	//iFinalVeloContactCaseAdv
		aTransferPackages[25].iChannel := iParameterSet;
		aTransferPackages[25].iAddressedTarget := 33;
		aTransferPackages[25].iIndex := 156;
		
	//iMeanPressureLevel
		aTransferPackages[26].iChannel := iParameterSet;
		aTransferPackages[26].iAddressedTarget := 33;
		aTransferPackages[26].iIndex := 184;
		
	// iThreshPosFollowError
		aTransferPackages[27].iChannel := iParameterSet;
		aTransferPackages[27].iAddressedTarget := 33;
		aTransferPackages[27].iIndex := 204;
		
	// iTreshVeloFollowError
		aTransferPackages[28].iChannel := iParameterSet;
		aTransferPackages[28].iAddressedTarget := 33;
		aTransferPackages[28].iIndex := 205;
		
	// iSoftStartFunction
		aTransferPackages[29].iChannel := iParameterSet;
		aTransferPackages[29].iAddressedTarget := 33;
		aTransferPackages[29].iIndex := 222;
		
	// iEndPositionMonitoring
		aTransferPackages[30].iChannel := iParameterSet;
		aTransferPackages[30].iAddressedTarget := 33;
		aTransferPackages[30].iIndex := 224;
		
	// xOptionPressureBuildUpIntoMechEndPos
		aTransferPackages[31].iChannel := iParameterSet;
		aTransferPackages[31].iAddressedTarget := 33;
		aTransferPackages[31].iIndex := 225;
		
	// iOptControllerGainRelative
		aTransferPackages[32].iChannel := iParameterSet;
		aTransferPackages[32].iAddressedTarget := 33;
		aTransferPackages[32].iIndex := 230;
		
	// iOptDampingOfSystemAbsolute
		aTransferPackages[33].iChannel := iParameterSet;
		aTransferPackages[33].iAddressedTarget := 33;
		aTransferPackages[33].iIndex := 231;
		
	// iOptPliabilityRelative
		aTransferPackages[34].iChannel := iParameterSet;
		aTransferPackages[34].iAddressedTarget := 33;
		aTransferPackages[34].iIndex := 232;
		
	// iOptReductionOfPilotControlRelative
		aTransferPackages[35].iChannel := iParameterSet;
		aTransferPackages[35].iAddressedTarget := 33;
		aTransferPackages[35].iIndex := 233;
		
	// iOptCoulombFritionInAccountRelative
		aTransferPackages[36].iChannel := iParameterSet;
		aTransferPackages[36].iAddressedTarget := 33;
		aTransferPackages[36].iIndex := 234;
		
	// define end of parameter list to be uploaded by setting all variables to 0 (end criterion for FB_Upload_Multiple_Parameters)
		aTransferPackages[37].iChannel := 0;
		aTransferPackages[37].iAddressedTarget := 0;
		aTransferPackages[37].iIndex := 0;
//-----------------------------------------------------------------------------------------------------------

// Read the current status of the the motion terminal
	fbreadbitsfromword(wData:= awBusDataFromVTEM[0], iStartBit:=0, iEndBit:= 5, iValue=> iCurrentValveMode, xError=> );				// read current valve mode
//-----------------------------------------------------------------------------------------------------------

// Transition: Aborting condition when xAbort is TRUE in all States except "IDLE" , "ABORTING" and "RESETTING"
	IF xAbort = TRUE AND NOT(iState = 10 AND xExecute = FALSE) AND iState <> 80 AND iState <> 100 THEN
		xStateChange := TRUE;	// Leaving current state
		iState := 80;	// Choosing next state, here: ABORTING
	END_IF
//-----------------------------------------------------------------------------------------------------------

// local state machine
	CASE iState OF
		10:	// IDLE
			// code that is executed only in the first cycle of this state
				IF xStateChange = TRUE THEN
					xStateChange := FALSE;
					iResponse := eTransferResponse.ready_for_new_transfer;
					xDone := FALSE;
					xError := FALSE;
					xBusy := FALSE;
					xAborted := FALSE;
				END_IF
			//-----------------------------------------------------------------------------------------------------------
			
			// code that is repeated every cycle in this state
				iCommandNumber := 0;
			//-----------------------------------------------------------------------------------------------------------
			
			// Transition
			IF xExecute = TRUE THEN
				xStateChange := TRUE;
				iState := 20;
			END_IF
			//-----------------------------------------------------------------------------------------------------------
		
		20:	// RESETTING VALVE MODE TO 61
			// code that is executed only in the first cycle of this state
				IF xStateChange = TRUE THEN
					xStateChange := FALSE;
					iResponse := eTransferResponse.preparing_transfer;
					xDone := FALSE;
					xError := FALSE;
					xBusy := TRUE;
					xAborted := FALSE;
				END_IF
			//-----------------------------------------------------------------------------------------------------------
			
			// code that is repeated every cycle in this state	
				IF iCurrentValveMode = 63 THEN
					iCommandNumber := 5;	// exit transfer mode
				ELSIF iCurrentValveMode <> 61 AND iCurrentValveMode <> 63 THEN
					iCommandNumber := 6;	// stop running motion apps
				END_IF 
			//-----------------------------------------------------------------------------------------------------------
			
			// Transition
				IF iCurrentValveMode = 61 THEN
					xStateChange := TRUE;	// Leave this state
					iState := 30;
					iCommandNumber := 30;			
				END_IF
			//-----------------------------------------------------------------------------------------------------------
		
		30:	// READING PARAMETER VALUES
			// code that is executed only in the first cycle of this state
				IF xStateChange = TRUE THEN
					xStateChange := FALSE;
					iResponse := eTransferResponse.transferring;
					xDone := FALSE;
					xError := FALSE;
					xBusy := TRUE;
					xAborted := FALSE;
				END_IF
			//-----------------------------------------------------------------------------------------------------------
			
			// code that is repeated every cycle in this state
				iCommandNumber := 30;		// read parameter values
			//-----------------------------------------------------------------------------------------------------------
			
			// Transition
				IF fbuploadMultipleParameters.xExecute = TRUE AND fbuploadMultipleParameters.xUploadDone = TRUE AND fbuploadMultipleParameters.xUploadError = FALSE THEN	// Upload Done
					xStateChange := TRUE;
					iState := 40;	// Write parameter values to outputs
				ELSIF fbuploadMultipleParameters.xExecute = TRUE AND fbuploadMultipleParameters.xUploadDone = FALSE AND fbuploadMultipleParameters.xUploadError = TRUE THEN	// Error during update
					xStateChange := TRUE;
					iState := 70;	// ERROR
					iResponse := fbuploadMultipleParameters.iResponse;
				END_IF
			//-----------------------------------------------------------------------------------------------------------
		
		40:	// WRITE PARAMETER VALUES TO OUTPUTS
			// code that is executed only in the first cycle of this state
				IF xStateChange = TRUE THEN
					xStateChange := FALSE;
					iResponse := eTransferResponse.transferring;
					xDone := FALSE;
					xError := FALSE;
					xBusy := TRUE;
					xAborted := FALSE;
				END_IF
			//-----------------------------------------------------------------------------------------------------------
			
			// code that is repeated every cycle in this state
				iTubingLengthAt2						:= aTransferPackages[0].iTransferValue;
				iTubingLengthAt4						:= aTransferPackages[1].iTransferValue;
				iTubingInnerDiameterAt2					:= aTransferPackages[2].iTransferValue;
				iTubingInnerDiameterAt4					:= aTransferPackages[3].iTransferValue;
				iDriveType								:= aTransferPackages[4].iTransferValue;
				iDriveStroke							:= aTransferPackages[5].iTransferValue;
				iInstallationPositionDrive				:= aTransferPackages[6].iTransferValue;
				iOffsetAxisZeroPoint					:= aTransferPackages[7].iTransferValue;
				iInPortFullStrokeMeas					:= aTransferPackages[8].iTransferValue;
				iInPortPartStrokeMeasRet				:= aTransferPackages[9].iTransferValue;
				iInPortPartStrokeMeasAdv				:= aTransferPackages[10].iTransferValue;
				iLoad									:= aTransferPackages[11].iTransferValue;
				iDampingTimeForTargetPositionReached	:= aTransferPackages[12].iTransferValue;
				iDurationOfThresholdExceedanceForError	:= aTransferPackages[13].iTransferValue;
				iToleranceForTargetPositionReached		:= aTransferPackages[14].iTransferValue;
				iMaxVelocityGeneral						:= aTransferPackages[15].iTransferValue;
				iMaxAcceleration						:= aTransferPackages[16].iTransferValue;
				iMaxDeceleration						:= aTransferPackages[17].iTransferValue;
				iMaxJerk								:= aTransferPackages[18].iTransferValue;
				iOffsetProjectZeroPoint					:= aTransferPackages[19].iTransferValue;
				iOffsetSoftLimitNegEndRet				:= aTransferPackages[20].iTransferValue;
				iOffsetSoftLimitPosEndAdv				:= aTransferPackages[21].iTransferValue;
				iDistTargPosWithConstVeloRet			:= aTransferPackages[22].iTransferValue;
				iFinalVeloContactCaseRet				:= aTransferPackages[23].iTransferValue;
				iDistTargPosWithConstVeloAdv			:= aTransferPackages[24].iTransferValue;
				iFinalVeloContactCaseAdv				:= aTransferPackages[25].iTransferValue;
				iMeanPressureLevel						:= aTransferPackages[26].iTransferValue;
				iThreshPosFollowError					:= aTransferPackages[27].iTransferValue;
				iTreshVeloFollowError					:= aTransferPackages[28].iTransferValue;
				iSoftStartFunction						:= aTransferPackages[29].iTransferValue;
				iEndPositionMonitoring					:= aTransferPackages[30].iTransferValue;
				xOptionPressureBuildUpIntoMechEndPos	:= INT_TO_BOOL(aTransferPackages[31].iTransferValue);
				iOptControllerGainRelative				:= aTransferPackages[32].iTransferValue;
				iOptDampingOfSystemAbsolute				:= aTransferPackages[33].iTransferValue;
				iOptPliabilityRelative					:= aTransferPackages[34].iTransferValue;
				iOptReductionOfPilotControlRelative		:= aTransferPackages[35].iTransferValue;
				iOptCoulombFritionInAccountRelative		:= aTransferPackages[36].iTransferValue;
			//-----------------------------------------------------------------------------------------------------------
			
			// Transition
				xStateChange := TRUE;
				iState := 50;
				iCommandNumber := 40;
			//-----------------------------------------------------------------------------------------------------------
		
		50:	// DONE
			// code that is executed only in the first cycle of this state
				IF xStateChange = TRUE THEN
					xStateChange := FALSE;
					iResponse := eTransferResponse.transfer_successful;
					xDone := TRUE;
					xError := FALSE;
					xBusy := FALSE;
					xAborted := FALSE;
				END_IF
			//-----------------------------------------------------------------------------------------------------------
			
			// code that is repeated every cycle in this state	
				IF fbuploadMultipleParameters.xExecute = FALSE  AND fbuploadMultipleParameters.xUploadDone = FALSE AND fbuploadMultipleParameters.xUploadError = FALSE AND iCurrentValveMode = 63 THEN		//FB_UploadMultipleParameters was reset
					iCommandNumber := 5;	// exit transfer mode
				END_IF
			//-----------------------------------------------------------------------------------------------------------
			
			// Transition
				IF fbuploadMultipleParameters.xExecute = FALSE  AND fbuploadMultipleParameters.xUploadDone = FALSE AND fbuploadMultipleParameters.xUploadError = FALSE AND xExecute = FALSE THEN
					xStateChange := TRUE;
					iState := 100;
				END_IF
			//-----------------------------------------------------------------------------------------------------------
			
		70:	// ERROR
			// code that is executed only in the first cycle of this state
				IF xStateChange = TRUE THEN
					xStateChange := FALSE;
					//iResponse := eTransferResponse.communication_failed;	// set within the transition of the last state
					xDone := FALSE;
					xError := TRUE;
					xBusy := FALSE;
					xAborted := FALSE;
				END_IF
			//-----------------------------------------------------------------------------------------------------------
			
			// code that is repeated every cycle in this state	
			//-----------------------------------------------------------------------------------------------------------
			
			// Transition
				IF xExecute = FALSE AND xAbort = FALSE THEN
					xStateChange := TRUE;
					iState := 100;
				END_IF
			//-----------------------------------------------------------------------------------------------------------
			
		80:	// ABORTING
			// code that is executed only in the first cycle of this state
				IF xStateChange = TRUE THEN
					xStateChange := FALSE;
					iResponse := eTransferResponse.aborting;
					xBusy := FALSE;
					xDone := FALSE;
					xError := FALSE;
					xAborted := TRUE;
				END_IF
			//-----------------------------------------------------------------------------------------------------------
			
			// code that is repeated every cycle in this state
				IF iCurrentValveMode = 63 THEN
					iCommandNumber := 5;	// exit transfer mode
				ELSIF iCurrentValveMode <> 61 AND iCurrentValveMode <> 63 THEN
					iCommandNumber := 6;	// stop running motion apps
				ELSE
					iCommandNumber := 0; 
				END_IF
			//-----------------------------------------------------------------------------------------------------------
			
			// Transition
				IF xAbort = FALSE AND xExecute = FALSE AND iCurrentValveMode = 61 THEN
					xStateChange := TRUE;
					iState := 100;
				END_IF
			//-----------------------------------------------------------------------------------------------------------

		100:	// RESETTING FUNCTION BLOCK AND VALVE
			// code that is executed only in the first cycle of this state
				IF xStateChange = TRUE THEN
					xStateChange := FALSE;
					iResponse := eTransferResponse.resetting;
					xDone := FALSE;
					xError := FALSE;
					xBusy := FALSE;
					xAborted := FALSE;
				END_IF
			//-----------------------------------------------------------------------------------------------------------
			
			// code that is repeated every cycle in this state	
				IF iCurrentValveMode = 63 THEN
					iCommandNumber := 5;	// exit transfer mode
				ELSIF iCurrentValveMode <> 61 AND iCurrentValveMode <> 63 THEN
					iCommandNumber := 6;	// stop running motion apps
				END_IF
				
				// reset funktion block fbreadmultipleparameters
				// not done via command number because this is used to reset valve
					fbuploadMultipleParameters(
						awBusDataFromVTEM:= awBusDataFromVTEM, 
						awBusDataToVTEM:= awBusDataToVTEM, 
						xExecute:= FALSE, 
						iResponse=> , 
						iCurrentValue=> , 
						xUploadDone=> , 
						xUploadError=> , 
						aTransferPackages:= aTransferPackages);
				
				// reset parameter outputs
					iParameterSet							:= 1;

					iTubingLengthAt2						:= 0;
					iTubingLengthAt4						:= 0;
					iTubingInnerDiameterAt2					:= 0;
					iTubingInnerDiameterAt4					:= 0;
					iDriveType								:= 0;
					iDriveStroke							:= 0;
					iInstallationPositionDrive				:= 0;
					iOffsetAxisZeroPoint					:= 0;
					iInPortFullStrokeMeas					:= 0;
					iInPortPartStrokeMeasRet				:= 0;
					iInPortPartStrokeMeasAdv				:= 0;
					iLoad									:= 0;
					iDampingTimeForTargetPositionReached	:= 0;
					iDurationOfThresholdExceedanceForError	:= 0;
					iToleranceForTargetPositionReached		:= 0;
					iMaxVelocityGeneral						:= 0;
					iMaxAcceleration						:= 0;
					iMaxDeceleration						:= 0;
					iMaxJerk								:= 0;
					iOffsetProjectZeroPoint					:= 0;
					iOffsetSoftLimitNegEndRet				:= 0;
					iOffsetSoftLimitPosEndAdv				:= 0;
					iDistTargPosWithConstVeloRet			:= 0;
					iFinalVeloContactCaseRet				:= 0;
					iDistTargPosWithConstVeloAdv			:= 0;
					iFinalVeloContactCaseAdv				:= 0;
					iMeanPressureLevel						:= 0;
					iThreshPosFollowError					:= 0;
					iTreshVeloFollowError					:= 0;
					iSoftStartFunction						:= 0;
					iEndPositionMonitoring					:= 0;
					xOptionPressureBuildUpIntoMechEndPos	:= 0;
					iOptControllerGainRelative				:= 0;
					iOptDampingOfSystemAbsolute				:= 0;
					iOptPliabilityRelative					:= 0;
					iOptReductionOfPilotControlRelative		:= 0;
					iOptCoulombFritionInAccountRelative		:= 0;
				
				// reset parameter array
					FOR iCounterResetArray := 0 TO 100 BY 1 DO
						aTransferPackages[iCounterResetArray].iChannel := 0;
						aTransferPackages[iCounterResetArray].iAddressedTarget := 0;
						aTransferPackages[iCounterResetArray].iIndex := 0;
						aTransferPackages[iCounterResetArray].iTransferValue := 0;
					END_FOR
					
					iCounterResetArray := 0;
					xFirstCycle := TRUE;
			//-----------------------------------------------------------------------------------------------------------
			
			// Transition
				IF iCurrentValveMode = 61 THEN
					iCommandNumber := 6; // Last command to send before the FB is in IDLE
					xStateChange := TRUE;
					iState := 10;
				END_IF
			//-----------------------------------------------------------------------------------------------------------
			
	END_CASE
//-----------------------------------------------------------------------------------------------------------

// Command section
	CASE iCommandNumber OF
		0:	// IDLE
			;
		
		5:	// EXIT TRANSFER MODE
			fbwritevaluetoword(iValue:=63, iStartBit:=0, iEndBit:=5, wDataWord:=awBusDataToVTEM[0], xError=> );							// Valve Mode = 63
			fbwritevaluetoword(iValue:=0, iStartBit:=6, iEndBit:=7, wDataWord:=awBusDataToVTEM[0], xError=> );							// 0 (unused)
			fbwritevaluetoword(iValue:=0, iStartBit:=8, iEndBit:=12, wDataWord:=awBusDataToVTEM[0], xError=> );							// Channel = 0 (ignored)
			fbwritevaluetoword(iValue:=3, iStartBit:=13, iEndBit:=15, wDataWord:=awBusDataToVTEM[0], xError=> );						// Transfer Control = 3 (Exit transfer mode)
			fbwritevaluetoword(iValue:=0, iStartBit:=0, iEndBit:=7, wDataWord:=awBusDataToVTEM[1], xError=> );							// Addressed Target = 0 (ignored)
			fbwritevaluetoword(iValue:=0, iStartBit:=8, iEndBit:=15, wDataWord:=awBusDataToVTEM[1], xError=> );							// Index = 0 (ignored)
			fbwritevaluetoword(iValue:=0, iStartBit:=0, iEndBit:=15, wDataWord:=awBusDataToVTEM[2], xError=> );							// Value = 0 (ignored)
			
		6:	// STOP RUNNING MOTION APP
			fbwritevaluetoword(iValue:=61, iStartBit:=0, iEndBit:=5, wDataWord:=awBusDataToVTEM[0], xError=> );							// Valve Mode = 61 (stop)
			fbwritevaluetoword(iValue:=0, iStartBit:=6, iEndBit:=7, wDataWord:=awBusDataToVTEM[0], xError=> );							// App Control = 0 (unused)
			fbwritevaluetoword(iValue:=0, iStartBit:=8, iEndBit:=15, wDataWord:=awBusDataToVTEM[0], xError=> );							// App Option = 0 (unused)
			fbwritevaluetoword(iValue:=0, iStartBit:=0, iEndBit:=15, wDataWord:=awBusDataToVTEM[1], xError=> );							// Setpoint Value 1 = 0 (unused)
			fbwritevaluetoword(iValue:=0, iStartBit:=0, iEndBit:=15, wDataWord:=awBusDataToVTEM[2], xError=> );							// Setpoint Value 2 = 0 (unused)
		
		30:	// RUN FB_UPLOADMULTIPLEPARAMETERS
			fbuploadMultipleParameters(
				awBusDataFromVTEM:= awBusDataFromVTEM, 
				awBusDataToVTEM:= awBusDataToVTEM, 
				xExecute:= TRUE, 
				iResponse=> , 
				iCurrentValue=> , 
				xUploadDone=> , 
				xUploadError=> , 
				aTransferPackages:= aTransferPackages);

		40:	// RESET FB_UPLOADMULTIPLEPARAMETERS
			fbuploadMultipleParameters(
				awBusDataFromVTEM:= awBusDataFromVTEM, 
				awBusDataToVTEM:= awBusDataToVTEM, 
				xExecute:= FALSE, 
				iResponse=> , 
				iCurrentValue=> , 
				xUploadDone=> , 
				xUploadError=> , 
				aTransferPackages:= aTransferPackages);
	END_CASE
//-----------------------------------------------------------------------------------------------------------

END_FUNCTION_BLOCK

// Transfermode/FB_Read_config_AI_Module
/// This function block can be used to upload the configuration of the analog input module on the Motion Terminal.
/// The specific parameters of this module are the outputs of this FB
/// The function block uses the transfer mode to read this configuration from the Motion Terminal
/// and indicates the state of the upload process at the output iResponse.

FUNCTION_BLOCK FB_Read_config_AI_Module
VAR_INPUT
	awBusDataFromVTEM 				: ARRAY [0..2] OF WORD;		// array of 3 words of process data received from the Motion Terminal
END_VAR
	
VAR_IN_OUT
	awBusDataToVTEM 				: ARRAY [0..2] OF WORD; 	// array of 3 words of process data sent to the Motion Terminal
END_VAR

VAR_INPUT
	xExecute 						: BOOL; 					// rising edge starts the reading process, falling edge resets the function block after reading is done
	xAbort							: BOOL;						// rising edge aborts the reading process
	iInputModuleNr					: INT;						// Number of the input module, counted from left to right beginning with 1
END_VAR                     		

VAR_OUTPUT                  		
	// sensor parameters
		iSensorTypePort0			: INT;						// ID of the sensor type, that is connected to the port 0 (0 = no sensor, 2001 = SDAP-MHS-M50, 2002 = SDAP-MHS-M100, 2003 = SDAP-MHS-M160, 2901 = custom position sensor 1, 2902 = custom position sensor 2, 2903 = custom position sensor 3, 3001 = SFAB-50U-…-2SA-…, 3002 = SFAB-200U-…-2SA-…, 3003 = SFAB-600U-…-2SA-…, 3004 = SFAB-1000U-…-2SA-…, 3101 = SFAH-50U-…-PNVBA-…, 3102 = SFAH-100U-…-PNVBA-…, 3103 = SFAH-200U-…-PNVBA-…, 3901 = custom flow sensor 1, 3902 = custom flow sensor 2, 3903 = custom flow sensor 3)
		iSensorOrientPort0			: INT;						// Orientation of the sensor that is connected to the port 0 (position sensor: 0 = risigng current level when advancing, 1 = falling current level when advancing; flow sensor: 0 = positive flow rate values "blowing", 1 = negative flow rate values "drawning")
		iSensorTypePort1			: INT;						// ID of the sensor type, that is connected to the port 1 (0 = no sensor, 2001 = SDAP-MHS-M50, 2002 = SDAP-MHS-M100, 2003 = SDAP-MHS-M160, 2901 = custom position sensor 1, 2902 = custom position sensor 2, 2903 = custom position sensor 3, 3001 = SFAB-50U-…-2SA-…, 3002 = SFAB-200U-…-2SA-…, 3003 = SFAB-600U-…-2SA-…, 3004 = SFAB-1000U-…-2SA-…, 3101 = SFAH-50U-…-PNVBA-…, 3102 = SFAH-100U-…-PNVBA-…, 3103 = SFAH-200U-…-PNVBA-…, 3901 = custom flow sensor 1, 3902 = custom flow sensor 2, 3903 = custom flow sensor 3)
		iSensorOrientPort1			: INT;						// Orientation of the sensor that is connected to the port 0 (position sensor: 0 = risigng current level when advancing, 1 = falling current level when advancing; flow sensor: 0 = positive flow rate values "blowing", 1 = negative flow rate values "drawning")
		iSensorTypePort2			: INT;						// ID of the sensor type, that is connected to the port 2 (0 = no sensor, 2001 = SDAP-MHS-M50, 2002 = SDAP-MHS-M100, 2003 = SDAP-MHS-M160, 2901 = custom position sensor 1, 2902 = custom position sensor 2, 2903 = custom position sensor 3, 3001 = SFAB-50U-…-2SA-…, 3002 = SFAB-200U-…-2SA-…, 3003 = SFAB-600U-…-2SA-…, 3004 = SFAB-1000U-…-2SA-…, 3101 = SFAH-50U-…-PNVBA-…, 3102 = SFAH-100U-…-PNVBA-…, 3103 = SFAH-200U-…-PNVBA-…, 3901 = custom flow sensor 1, 3902 = custom flow sensor 2, 3903 = custom flow sensor 3)
		iSensorOrientPort2			: INT;						// Orientation of the sensor that is connected to the port 0 (position sensor: 0 = risigng current level when advancing, 1 = falling current level when advancing; flow sensor: 0 = positive flow rate values "blowing", 1 = negative flow rate values "drawning")
		iSensorTypePort3			: INT;						// ID of the sensor type, that is connected to the port 3 (0 = no sensor, 2001 = SDAP-MHS-M50, 2002 = SDAP-MHS-M100, 2003 = SDAP-MHS-M160, 2901 = custom position sensor 1, 2902 = custom position sensor 2, 2903 = custom position sensor 3, 3001 = SFAB-50U-…-2SA-…, 3002 = SFAB-200U-…-2SA-…, 3003 = SFAB-600U-…-2SA-…, 3004 = SFAB-1000U-…-2SA-…, 3101 = SFAH-50U-…-PNVBA-…, 3102 = SFAH-100U-…-PNVBA-…, 3103 = SFAH-200U-…-PNVBA-…, 3901 = custom flow sensor 1, 3902 = custom flow sensor 2, 3903 = custom flow sensor 3)
		iSensorOrientPort3			: INT;						// Orientation of the sensor that is connected to the port 0 (position sensor: 0 = risigng current level when advancing, 1 = falling current level when advancing; flow sensor: 0 = positive flow rate values "blowing", 1 = negative flow rate values "drawning")
		iSensorTypePort4			: INT;						// ID of the sensor type, that is connected to the port 4 (0 = no sensor, 2001 = SDAP-MHS-M50, 2002 = SDAP-MHS-M100, 2003 = SDAP-MHS-M160, 2901 = custom position sensor 1, 2902 = custom position sensor 2, 2903 = custom position sensor 3, 3001 = SFAB-50U-…-2SA-…, 3002 = SFAB-200U-…-2SA-…, 3003 = SFAB-600U-…-2SA-…, 3004 = SFAB-1000U-…-2SA-…, 3101 = SFAH-50U-…-PNVBA-…, 3102 = SFAH-100U-…-PNVBA-…, 3103 = SFAH-200U-…-PNVBA-…, 3901 = custom flow sensor 1, 3902 = custom flow sensor 2, 3903 = custom flow sensor 3)
		iSensorOrientPort4			: INT;						// Orientation of the sensor that is connected to the port 0 (position sensor: 0 = risigng current level when advancing, 1 = falling current level when advancing; flow sensor: 0 = positive flow rate values "blowing", 1 = negative flow rate values "drawning")
		iSensorTypePort5			: INT;						// ID of the sensor type, that is connected to the port 5 (0 = no sensor, 2001 = SDAP-MHS-M50, 2002 = SDAP-MHS-M100, 2003 = SDAP-MHS-M160, 2901 = custom position sensor 1, 2902 = custom position sensor 2, 2903 = custom position sensor 3, 3001 = SFAB-50U-…-2SA-…, 3002 = SFAB-200U-…-2SA-…, 3003 = SFAB-600U-…-2SA-…, 3004 = SFAB-1000U-…-2SA-…, 3101 = SFAH-50U-…-PNVBA-…, 3102 = SFAH-100U-…-PNVBA-…, 3103 = SFAH-200U-…-PNVBA-…, 3901 = custom flow sensor 1, 3902 = custom flow sensor 2, 3903 = custom flow sensor 3)
		iSensorOrientPort5			: INT;						// Orientation of the sensor that is connected to the port 0 (position sensor: 0 = risigng current level when advancing, 1 = falling current level when advancing; flow sensor: 0 = positive flow rate values "blowing", 1 = negative flow rate values "drawning")
		iSensorTypePort6			: INT;						// ID of the sensor type, that is connected to the port 6 (0 = no sensor, 2001 = SDAP-MHS-M50, 2002 = SDAP-MHS-M100, 2003 = SDAP-MHS-M160, 2901 = custom position sensor 1, 2902 = custom position sensor 2, 2903 = custom position sensor 3, 3001 = SFAB-50U-…-2SA-…, 3002 = SFAB-200U-…-2SA-…, 3003 = SFAB-600U-…-2SA-…, 3004 = SFAB-1000U-…-2SA-…, 3101 = SFAH-50U-…-PNVBA-…, 3102 = SFAH-100U-…-PNVBA-…, 3103 = SFAH-200U-…-PNVBA-…, 3901 = custom flow sensor 1, 3902 = custom flow sensor 2, 3903 = custom flow sensor 3)
		iSensorOrientPort6			: INT;						// Orientation of the sensor that is connected to the port 0 (position sensor: 0 = risigng current level when advancing, 1 = falling current level when advancing; flow sensor: 0 = positive flow rate values "blowing", 1 = negative flow rate values "drawning")
		iSensorTypePort7			: INT;						// ID of the sensor type, that is connected to the port 7 (0 = no sensor, 2001 = SDAP-MHS-M50, 2002 = SDAP-MHS-M100, 2003 = SDAP-MHS-M160, 2901 = custom position sensor 1, 2902 = custom position sensor 2, 2903 = custom position sensor 3, 3001 = SFAB-50U-…-2SA-…, 3002 = SFAB-200U-…-2SA-…, 3003 = SFAB-600U-…-2SA-…, 3004 = SFAB-1000U-…-2SA-…, 3101 = SFAH-50U-…-PNVBA-…, 3102 = SFAH-100U-…-PNVBA-…, 3103 = SFAH-200U-…-PNVBA-…, 3901 = custom flow sensor 1, 3902 = custom flow sensor 2, 3903 = custom flow sensor 3)
		iSensorOrientPort7			: INT;						// Orientation of the sensor that is connected to the port 0 (position sensor: 0 = risigng current level when advancing, 1 = falling current level when advancing; flow sensor: 0 = positive flow rate values "blowing", 1 = negative flow rate values "drawning")
		
	// function block response
		iResponse 					: eTransferResponse; 		// returns the status of the upload process
		xBusy						: BOOL;						// TRUE as long as the upload process is running
		xDone 						: BOOL; 					// indicates whether the upload was successfull
		xError 						: BOOL; 					// indicates whether an error occurred during the transfer
		xAborted					: BOOL;						// TRUE if the function block was canceled by xAbort	
END_VAR

VAR
	iState							: INT := 10;
	xStateChange					: BOOL;
	iCommandNumber					: INT;
	xFirstCycle						: BOOL := TRUE;				// indicator for the first cycle of the function block
	iInputModuleNrFC				: INT;						// value on input iInputModuleNr during first cycle
	
	aTransferPackages				: ARRAY [0..100] OF stTransferPackage;
	fbreadbitsfromword				: FB_Read_Bits_From_Word;
	fbuploadMultipleParameters 		: FB_Upload_Multiple_Parameters;
	fbWriteValueToWord 				: FB_Write_Value_To_Word;

	iCounterResetArray				: INT;

	iCurrentValveMode				: INT;						//
END_VAR

(*****************************************************************************************************

Festo SE & Co. KG, Esslingen
Copyright (c) 2021. All rights reserved.

Product:            Motion Terminal VTEM
Description:        Function block to upload the analog module parameters from the Motion Terminal

Object version:     2.00
Last change:        2021-07
======================================================================================================
                                       H I S T O R Y
======================================================================================================
Version:            2.00
Date:               2021-07
Change/Activity:    - created (#3872357)
Release:            3.5.7.237 (CODESYS 3.5.7.2, Lib version 3.7)
Author:             JEBU
======================================================================================================

*****************************************************************************************************)

// pre-check of the value for the parameter set
	IF xExecute = TRUE AND (iInputModuleNr < 1 OR iInputModuleNr > 2) THEN		// invalid input for the module number
		xDone := FALSE; 
		xError := TRUE; 
		iResponse := eTransferResponse.invalid_module_number;
		xStateChange := TRUE;
		iState := 70;	// ERROR
	END_IF
//-----------------------------------------------------------------------------------------------------------

// check if iInputModuleNr was changed
	IF xExecute = TRUE AND xFirstCycle = TRUE THEN
		xFirstCycle := FALSE;
		iInputModuleNrFC := iInputModuleNr;
	END_IF
	
	IF xExecute = TRUE AND iInputModuleNr <> iInputModuleNrFC THEN
		xStateChange := TRUE;
		iState := 70;
		iResponse := eTransferResponse.FB_needs_rising_edge_xExecute;
	END_IF
//-----------------------------------------------------------------------------------------------------------

// WRITE PARAMETER INDICES INTO ARRAY
	// ID of sensor at port 0
		aTransferPackages[0].iChannel := 16;
		aTransferPackages[0].iAddressedTarget := iInputModuleNr;
		aTransferPackages[0].iIndex := 1;
		
	// Orientation of the sensor at port 0
		aTransferPackages[1].iChannel := 16;
		aTransferPackages[1].iAddressedTarget := iInputModuleNr;
		aTransferPackages[1].iIndex := 2;
		
	// ID of sensor at port 1
		aTransferPackages[2].iChannel := 16;
		aTransferPackages[2].iAddressedTarget := iInputModuleNr;
		aTransferPackages[2].iIndex := 31;
		
	// Orientation of the sensor at port 1
		aTransferPackages[3].iChannel := 16;
		aTransferPackages[3].iAddressedTarget := iInputModuleNr;
		aTransferPackages[3].iIndex := 32;
		
	// ID of sensor at port 2
		aTransferPackages[4].iChannel := 16;
		aTransferPackages[4].iAddressedTarget := iInputModuleNr;
		aTransferPackages[4].iIndex := 61;
		
	// Orientation of the sensor at port 2
		aTransferPackages[5].iChannel := 16;
		aTransferPackages[5].iAddressedTarget := iInputModuleNr;
		aTransferPackages[5].iIndex := 62;
		
	// ID of sensor at port 3
		aTransferPackages[6].iChannel := 16;
		aTransferPackages[6].iAddressedTarget := iInputModuleNr;
		aTransferPackages[6].iIndex := 91;
		
	// Orientation of the sensor at port 3
		aTransferPackages[7].iChannel := 16;
		aTransferPackages[7].iAddressedTarget := iInputModuleNr;
		aTransferPackages[7].iIndex := 92;
		
	// ID of sensor at port 4
		aTransferPackages[8].iChannel := 16;
		aTransferPackages[8].iAddressedTarget := iInputModuleNr;
		aTransferPackages[8].iIndex := 121;
		
	// Orientation of the sensor at port 4
		aTransferPackages[9].iChannel := 16;
		aTransferPackages[9].iAddressedTarget := iInputModuleNr;
		aTransferPackages[9].iIndex := 122;
		
	// ID of sensor at port 5
		aTransferPackages[10].iChannel := 16;
		aTransferPackages[10].iAddressedTarget := iInputModuleNr;
		aTransferPackages[10].iIndex := 151;
		
	// Orientation of the sensor at port 5
		aTransferPackages[11].iChannel := 16;
		aTransferPackages[11].iAddressedTarget := iInputModuleNr;
		aTransferPackages[11].iIndex := 152;
		
	// ID of sensor at port 6
		aTransferPackages[12].iChannel := 16;
		aTransferPackages[12].iAddressedTarget := iInputModuleNr;
		aTransferPackages[12].iIndex := 181;
		
	// Orientation of the sensor at port 6
		aTransferPackages[13].iChannel := 16;
		aTransferPackages[13].iAddressedTarget := iInputModuleNr;
		aTransferPackages[13].iIndex := 182;
		
	// ID of sensor at port 7
		aTransferPackages[14].iChannel := 16;
		aTransferPackages[14].iAddressedTarget := iInputModuleNr;
		aTransferPackages[14].iIndex := 211;
		
	// Orientation of the sensor at port 7
		aTransferPackages[15].iChannel := 16;
		aTransferPackages[15].iAddressedTarget := iInputModuleNr;
		aTransferPackages[15].iIndex := 212;
		
	// define end of parameter list to be uploaded by setting all variables to 0 (end criterion for FB_Upload_Multiple_Parameters)
		aTransferPackages[16].iChannel := 0;
		aTransferPackages[16].iAddressedTarget := 0;
		aTransferPackages[16].iIndex := 0;
//-----------------------------------------------------------------------------------------------------------

// Read the current status of the the motion terminal
	fbreadbitsfromword(wData:= awBusDataFromVTEM[0], iStartBit:=0, iEndBit:= 5, iValue=> iCurrentValveMode, xError=> );				// read current valve mode
//-----------------------------------------------------------------------------------------------------------

// Transition: Aborting condition when xAbort is TRUE in all States except "IDLE" , "ABORTING" and "RESETTING"
	IF xAbort = TRUE AND NOT(iState = 10 AND xExecute = FALSE) AND iState <> 80 AND iState <> 100 THEN
		xStateChange := TRUE;	// Leaving current state
		iState := 80;	// Choosing next state, here: ABORTING
	END_IF
//-----------------------------------------------------------------------------------------------------------

// local state machine
	CASE iState OF
		10:	// IDLE
			// code that is executed only in the first cycle of this state
				IF xStateChange = TRUE THEN
					xStateChange := FALSE;
					iResponse := eTransferResponse.ready_for_new_transfer;
					xDone := FALSE;
					xError := FALSE;
					xBusy := FALSE;
					xAborted := FALSE;
				END_IF
			//-----------------------------------------------------------------------------------------------------------
			
			// code that is repeated every cycle in this state
				iCommandNumber := 0;
			//-----------------------------------------------------------------------------------------------------------
			
			// Transition
			IF xExecute = TRUE THEN
				xStateChange := TRUE;
				iState := 20;
			END_IF
			//-----------------------------------------------------------------------------------------------------------
		
		20:	// RESETTING VALVE MODE TO 61
			// code that is executed only in the first cycle of this state
				IF xStateChange = TRUE THEN
					xStateChange := FALSE;
					iResponse := eTransferResponse.preparing_transfer;
					xDone := FALSE;
					xError := FALSE;
					xBusy := TRUE;
					xAborted := FALSE;
				END_IF
			//-----------------------------------------------------------------------------------------------------------
			
			// code that is repeated every cycle in this state	
				IF iCurrentValveMode = 63 THEN
					iCommandNumber := 5;	// exit transfer mode
				ELSIF iCurrentValveMode <> 61 AND iCurrentValveMode <> 63 THEN
					iCommandNumber := 6;	// stop running motion apps
				END_IF 
			//-----------------------------------------------------------------------------------------------------------
			
			// Transition
				IF iCurrentValveMode = 61 THEN
					xStateChange := TRUE;	// Leave this state
					iState := 30;
					iCommandNumber := 30;			
				END_IF
			//-----------------------------------------------------------------------------------------------------------
		
		30:	// READING PARAMETER VALUES
			// code that is executed only in the first cycle of this state
				IF xStateChange = TRUE THEN
					xStateChange := FALSE;
					iResponse := eTransferResponse.transferring;
					xDone := FALSE;
					xError := FALSE;
					xBusy := TRUE;
					xAborted := FALSE;
				END_IF
			//-----------------------------------------------------------------------------------------------------------
			
			// code that is repeated every cycle in this state
				iCommandNumber := 30;		// read parameter values
			//-----------------------------------------------------------------------------------------------------------
			
			// Transition
				IF fbuploadMultipleParameters.xExecute = TRUE AND fbuploadMultipleParameters.xUploadDone = TRUE AND fbuploadMultipleParameters.xUploadError = FALSE THEN	// Upload Done
					xStateChange := TRUE;
					iState := 40;	// Write parameter values to outputs
				ELSIF fbuploadMultipleParameters.xExecute = TRUE AND fbuploadMultipleParameters.xUploadDone = FALSE AND fbuploadMultipleParameters.xUploadError = TRUE THEN	// Error during update
					xStateChange := TRUE;
					iState := 70;	// ERROR
					iResponse := fbuploadMultipleParameters.iResponse;
				END_IF
			//-----------------------------------------------------------------------------------------------------------
		
		40:	// WRITE PARAMETER VALUES TO OUTPUTS
			// code that is executed only in the first cycle of this state
				IF xStateChange = TRUE THEN
					xStateChange := FALSE;
					iResponse := eTransferResponse.transferring;
					xDone := FALSE;
					xError := FALSE;
					xBusy := TRUE;
					xAborted := FALSE;
				END_IF
			//-----------------------------------------------------------------------------------------------------------
			
			// code that is repeated every cycle in this state
				iSensorTypePort0		:= aTransferPackages[0].iTransferValue;
				iSensorOrientPort0		:= aTransferPackages[1].iTransferValue;
				iSensorTypePort1		:= aTransferPackages[2].iTransferValue;
				iSensorOrientPort1		:= aTransferPackages[3].iTransferValue;
				iSensorTypePort2		:= aTransferPackages[4].iTransferValue;
				iSensorOrientPort2		:= aTransferPackages[5].iTransferValue;
				iSensorTypePort3		:= aTransferPackages[6].iTransferValue;
				iSensorOrientPort3		:= aTransferPackages[7].iTransferValue;
				iSensorTypePort4		:= aTransferPackages[8].iTransferValue;
				iSensorOrientPort4		:= aTransferPackages[9].iTransferValue;
				iSensorTypePort5		:= aTransferPackages[10].iTransferValue;
				iSensorOrientPort5		:= aTransferPackages[11].iTransferValue;
				iSensorTypePort6		:= aTransferPackages[12].iTransferValue;
				iSensorOrientPort6		:= aTransferPackages[13].iTransferValue;
				iSensorTypePort7		:= aTransferPackages[14].iTransferValue;
				iSensorOrientPort7		:= aTransferPackages[15].iTransferValue;
			//-----------------------------------------------------------------------------------------------------------
			
			// Transition
				xStateChange := TRUE;
				iState := 50;
				iCommandNumber := 40;
			//-----------------------------------------------------------------------------------------------------------
		
		50:	// DONE
			// code that is executed only in the first cycle of this state
				IF xStateChange = TRUE THEN
					xStateChange := FALSE;
					iResponse := eTransferResponse.transfer_successful;
					xDone := TRUE;
					xError := FALSE;
					xBusy := FALSE;
					xAborted := FALSE;
				END_IF
			//-----------------------------------------------------------------------------------------------------------
			
			// code that is repeated every cycle in this state	
				IF fbuploadMultipleParameters.xExecute = FALSE  AND fbuploadMultipleParameters.xUploadDone = FALSE AND fbuploadMultipleParameters.xUploadError = FALSE AND iCurrentValveMode = 63 THEN		//FB_UploadMultipleParameters was reset
					iCommandNumber := 5;	// exit transfer mode
				END_IF
			//-----------------------------------------------------------------------------------------------------------
			
			// Transition
				IF fbuploadMultipleParameters.xExecute = FALSE  AND fbuploadMultipleParameters.xUploadDone = FALSE AND fbuploadMultipleParameters.xUploadError = FALSE AND xExecute = FALSE THEN
					xStateChange := TRUE;
					iState := 100;
				END_IF
			//-----------------------------------------------------------------------------------------------------------
			
		70:	// ERROR
			// code that is executed only in the first cycle of this state
				IF xStateChange = TRUE THEN
					xStateChange := FALSE;
					//iResponse := ;	// set within the transition of the last state
					xDone := FALSE;
					xError := TRUE;
					xBusy := FALSE;
					xAborted := FALSE;
				END_IF
			//-----------------------------------------------------------------------------------------------------------
			
			// code that is repeated every cycle in this state
				IF iResponse = eTransferResponse.invalid_Index THEN
					iResponse := eTransferResponse.invalid_module_number;
				END_IF
			//-----------------------------------------------------------------------------------------------------------
			
			// Transition
				IF xExecute = FALSE AND xAbort = FALSE THEN
					xStateChange := TRUE;
					iState := 100;
				END_IF
			//-----------------------------------------------------------------------------------------------------------
			
		80:	// ABORTING
			// code that is executed only in the first cycle of this state
				IF xStateChange = TRUE THEN
					xStateChange := FALSE;
					iResponse := eTransferResponse.aborting;
					xBusy := FALSE;
					xDone := FALSE;
					xError := FALSE;
					xAborted := TRUE;
				END_IF
			//-----------------------------------------------------------------------------------------------------------
			
			// code that is repeated every cycle in this state
				IF iCurrentValveMode = 63 THEN
					iCommandNumber := 5;	// exit transfer mode
				ELSIF iCurrentValveMode <> 61 AND iCurrentValveMode <> 63 THEN
					iCommandNumber := 6;	// stop running motion apps
				ELSE
					iCommandNumber := 0; 
				END_IF
			//-----------------------------------------------------------------------------------------------------------
			
			// Transition
				IF xAbort = FALSE AND xExecute = FALSE AND iCurrentValveMode = 61 THEN
					xStateChange := TRUE;
					iState := 100;
				END_IF
			//-----------------------------------------------------------------------------------------------------------

		100:	// RESETTING FUNCTION BLOCK AND VALVE
			// code that is executed only in the first cycle of this state
				IF xStateChange = TRUE THEN
					xStateChange := FALSE;
					iResponse := eTransferResponse.resetting;
					xDone := FALSE;
					xError := FALSE;
					xBusy := FALSE;
					xAborted := FALSE;
				END_IF
			//-----------------------------------------------------------------------------------------------------------
			
			// code that is repeated every cycle in this state	
				IF iCurrentValveMode = 63 THEN
					iCommandNumber := 5;	// exit transfer mode
				ELSIF iCurrentValveMode <> 61 AND iCurrentValveMode <> 63 THEN
					iCommandNumber := 6;	// stop running motion apps
				END_IF
				
				// reset funktion block fbreadmultipleparameters
				// not done via command number because this is used to reset valve
					fbuploadMultipleParameters(
						awBusDataFromVTEM:= awBusDataFromVTEM, 
						awBusDataToVTEM:= awBusDataToVTEM, 
						xExecute:= FALSE, 
						iResponse=> , 
						iCurrentValue=> , 
						xUploadDone=> , 
						xUploadError=> , 
						aTransferPackages:= aTransferPackages);

				// reset parameter outputs
					iInputModuleNr			:= 0;

					iSensorTypePort0		:= 0;
					iSensorOrientPort0		:= 0;
					iSensorTypePort1		:= 0;
					iSensorOrientPort1		:= 0;
					iSensorTypePort2		:= 0;
					iSensorOrientPort2		:= 0;
					iSensorTypePort3		:= 0;
					iSensorOrientPort3		:= 0;
					iSensorTypePort4		:= 0;
					iSensorOrientPort4		:= 0;
					iSensorTypePort5		:= 0;
					iSensorOrientPort5		:= 0;
					iSensorTypePort6		:= 0;
					iSensorOrientPort6		:= 0;
					iSensorTypePort7		:= 0;
					iSensorOrientPort7		:= 0;
				
				// reset parameter array
					FOR iCounterResetArray := 0 TO 100 BY 1 DO
						aTransferPackages[iCounterResetArray].iChannel := 0;
						aTransferPackages[iCounterResetArray].iAddressedTarget := 0;
						aTransferPackages[iCounterResetArray].iIndex := 0;
						aTransferPackages[iCounterResetArray].iTransferValue := 0;
					END_FOR
					
					iCounterResetArray := 0;
					xFirstCycle := TRUE;
			//-----------------------------------------------------------------------------------------------------------
			
			// Transition
				IF iCurrentValveMode = 61 THEN
					iCommandNumber := 6; // Last command to send before the FB is in IDLE
					xStateChange := TRUE;
					iState := 10;
				END_IF
			//-----------------------------------------------------------------------------------------------------------
			
	END_CASE
//-----------------------------------------------------------------------------------------------------------

// Command section
	CASE iCommandNumber OF
		0:	// IDLE
			;
		
		5:	// EXIT TRANSFER MODE
			fbwritevaluetoword(iValue:=63, iStartBit:=0, iEndBit:=5, wDataWord:=awBusDataToVTEM[0], xError=> );							// Valve Mode = 63
			fbwritevaluetoword(iValue:=0, iStartBit:=6, iEndBit:=7, wDataWord:=awBusDataToVTEM[0], xError=> );							// 0 (unused)
			fbwritevaluetoword(iValue:=0, iStartBit:=8, iEndBit:=12, wDataWord:=awBusDataToVTEM[0], xError=> );							// Channel = 0 (ignored)
			fbwritevaluetoword(iValue:=3, iStartBit:=13, iEndBit:=15, wDataWord:=awBusDataToVTEM[0], xError=> );						// Transfer Control = 3 (Exit transfer mode)
			fbwritevaluetoword(iValue:=0, iStartBit:=0, iEndBit:=7, wDataWord:=awBusDataToVTEM[1], xError=> );							// Addressed Target = 0 (ignored)
			fbwritevaluetoword(iValue:=0, iStartBit:=8, iEndBit:=15, wDataWord:=awBusDataToVTEM[1], xError=> );							// Index = 0 (ignored)
			fbwritevaluetoword(iValue:=0, iStartBit:=0, iEndBit:=15, wDataWord:=awBusDataToVTEM[2], xError=> );							// Value = 0 (ignored)
			
		6:	// STOP RUNNING MOTION APP
			fbwritevaluetoword(iValue:=61, iStartBit:=0, iEndBit:=5, wDataWord:=awBusDataToVTEM[0], xError=> );							// Valve Mode = 61 (stop)
			fbwritevaluetoword(iValue:=0, iStartBit:=6, iEndBit:=7, wDataWord:=awBusDataToVTEM[0], xError=> );							// App Control = 0 (unused)
			fbwritevaluetoword(iValue:=0, iStartBit:=8, iEndBit:=15, wDataWord:=awBusDataToVTEM[0], xError=> );							// App Option = 0 (unused)
			fbwritevaluetoword(iValue:=0, iStartBit:=0, iEndBit:=15, wDataWord:=awBusDataToVTEM[1], xError=> );							// Setpoint Value 1 = 0 (unused)
			fbwritevaluetoword(iValue:=0, iStartBit:=0, iEndBit:=15, wDataWord:=awBusDataToVTEM[2], xError=> );							// Setpoint Value 2 = 0 (unused)
		
		30:	// RUN FB_UPLOADMULTIPLEPARAMETERS
			fbuploadMultipleParameters(
				awBusDataFromVTEM:= awBusDataFromVTEM, 
				awBusDataToVTEM:= awBusDataToVTEM, 
				xExecute:= TRUE, 
				iResponse=> , 
				iCurrentValue=> , 
				xUploadDone=> , 
				xUploadError=> , 
				aTransferPackages:= aTransferPackages);

		40:	// RESET FB_UPLOADMULTIPLEPARAMETERS
			fbuploadMultipleParameters(
				awBusDataFromVTEM:= awBusDataFromVTEM, 
				awBusDataToVTEM:= awBusDataToVTEM, 
				xExecute:= FALSE, 
				iResponse=> , 
				iCurrentValue=> , 
				xUploadDone=> , 
				xUploadError=> , 
				aTransferPackages:= aTransferPackages);
	END_CASE
//-----------------------------------------------------------------------------------------------------------

END_FUNCTION_BLOCK

// Transfermode/FB_Read_config_DI_Module
/// This function block can be used to upload the configuration of the digital input module on the Motion Terminal.
/// The specific parameters of this module are the outputs of this FB
/// The function block uses the transfer mode to read this configuration from the Motion Terminal
/// and indicates the state of the upload process at the output iResponse.

FUNCTION_BLOCK FB_Read_config_DI_Module
VAR_INPUT
	awBusDataFromVTEM 				: ARRAY [0..2] OF WORD;		// array of 3 words of process data received from the Motion Terminal
END_VAR
	
VAR_IN_OUT
	awBusDataToVTEM 				: ARRAY [0..2] OF WORD; 	// array of 3 words of process data sent to the Motion Terminal
END_VAR

VAR_INPUT
	xExecute 						: BOOL; 					// rising edge starts the reading process, falling edge resets the function block after reading is done
	xAbort							: BOOL;						// rising edge aborts the reading process
	iInputModuleNr					: INT;						// Number of the input module, counted from left to right beginning with 1
END_VAR                     		

VAR_OUTPUT                  		
	// sensor parameters
		iSensorTypePort0			: INT;						// ID of the sensor type, that is connected to the port 0 (0 = no sensor, 2001 = SDAP-MHS-M50, 2002 = SDAP-MHS-M100, 2003 = SDAP-MHS-M160, 2901 = custom position sensor 1, 2902 = custom position sensor 2, 2903 = custom position sensor 3, 3001 = SFAB-50U-…-2SA-…, 3002 = SFAB-200U-…-2SA-…, 3003 = SFAB-600U-…-2SA-…, 3004 = SFAB-1000U-…-2SA-…, 3101 = SFAH-50U-…-PNVBA-…, 3102 = SFAH-100U-…-PNVBA-…, 3103 = SFAH-200U-…-PNVBA-…, 3901 = custom flow sensor 1, 3902 = custom flow sensor 2, 3903 = custom flow sensor 3)
		iSensorTypePort1			: INT;						// ID of the sensor type, that is connected to the port 1 (0 = no sensor, 2001 = SDAP-MHS-M50, 2002 = SDAP-MHS-M100, 2003 = SDAP-MHS-M160, 2901 = custom position sensor 1, 2902 = custom position sensor 2, 2903 = custom position sensor 3, 3001 = SFAB-50U-…-2SA-…, 3002 = SFAB-200U-…-2SA-…, 3003 = SFAB-600U-…-2SA-…, 3004 = SFAB-1000U-…-2SA-…, 3101 = SFAH-50U-…-PNVBA-…, 3102 = SFAH-100U-…-PNVBA-…, 3103 = SFAH-200U-…-PNVBA-…, 3901 = custom flow sensor 1, 3902 = custom flow sensor 2, 3903 = custom flow sensor 3)
		iSensorTypePort2			: INT;						// ID of the sensor type, that is connected to the port 2 (0 = no sensor, 2001 = SDAP-MHS-M50, 2002 = SDAP-MHS-M100, 2003 = SDAP-MHS-M160, 2901 = custom position sensor 1, 2902 = custom position sensor 2, 2903 = custom position sensor 3, 3001 = SFAB-50U-…-2SA-…, 3002 = SFAB-200U-…-2SA-…, 3003 = SFAB-600U-…-2SA-…, 3004 = SFAB-1000U-…-2SA-…, 3101 = SFAH-50U-…-PNVBA-…, 3102 = SFAH-100U-…-PNVBA-…, 3103 = SFAH-200U-…-PNVBA-…, 3901 = custom flow sensor 1, 3902 = custom flow sensor 2, 3903 = custom flow sensor 3)
		iSensorTypePort3			: INT;						// ID of the sensor type, that is connected to the port 3 (0 = no sensor, 2001 = SDAP-MHS-M50, 2002 = SDAP-MHS-M100, 2003 = SDAP-MHS-M160, 2901 = custom position sensor 1, 2902 = custom position sensor 2, 2903 = custom position sensor 3, 3001 = SFAB-50U-…-2SA-…, 3002 = SFAB-200U-…-2SA-…, 3003 = SFAB-600U-…-2SA-…, 3004 = SFAB-1000U-…-2SA-…, 3101 = SFAH-50U-…-PNVBA-…, 3102 = SFAH-100U-…-PNVBA-…, 3103 = SFAH-200U-…-PNVBA-…, 3901 = custom flow sensor 1, 3902 = custom flow sensor 2, 3903 = custom flow sensor 3)
		iSensorTypePort4			: INT;						// ID of the sensor type, that is connected to the port 4 (0 = no sensor, 2001 = SDAP-MHS-M50, 2002 = SDAP-MHS-M100, 2003 = SDAP-MHS-M160, 2901 = custom position sensor 1, 2902 = custom position sensor 2, 2903 = custom position sensor 3, 3001 = SFAB-50U-…-2SA-…, 3002 = SFAB-200U-…-2SA-…, 3003 = SFAB-600U-…-2SA-…, 3004 = SFAB-1000U-…-2SA-…, 3101 = SFAH-50U-…-PNVBA-…, 3102 = SFAH-100U-…-PNVBA-…, 3103 = SFAH-200U-…-PNVBA-…, 3901 = custom flow sensor 1, 3902 = custom flow sensor 2, 3903 = custom flow sensor 3)
		iSensorTypePort5			: INT;						// ID of the sensor type, that is connected to the port 5 (0 = no sensor, 2001 = SDAP-MHS-M50, 2002 = SDAP-MHS-M100, 2003 = SDAP-MHS-M160, 2901 = custom position sensor 1, 2902 = custom position sensor 2, 2903 = custom position sensor 3, 3001 = SFAB-50U-…-2SA-…, 3002 = SFAB-200U-…-2SA-…, 3003 = SFAB-600U-…-2SA-…, 3004 = SFAB-1000U-…-2SA-…, 3101 = SFAH-50U-…-PNVBA-…, 3102 = SFAH-100U-…-PNVBA-…, 3103 = SFAH-200U-…-PNVBA-…, 3901 = custom flow sensor 1, 3902 = custom flow sensor 2, 3903 = custom flow sensor 3)
		iSensorTypePort6			: INT;						// ID of the sensor type, that is connected to the port 6 (0 = no sensor, 2001 = SDAP-MHS-M50, 2002 = SDAP-MHS-M100, 2003 = SDAP-MHS-M160, 2901 = custom position sensor 1, 2902 = custom position sensor 2, 2903 = custom position sensor 3, 3001 = SFAB-50U-…-2SA-…, 3002 = SFAB-200U-…-2SA-…, 3003 = SFAB-600U-…-2SA-…, 3004 = SFAB-1000U-…-2SA-…, 3101 = SFAH-50U-…-PNVBA-…, 3102 = SFAH-100U-…-PNVBA-…, 3103 = SFAH-200U-…-PNVBA-…, 3901 = custom flow sensor 1, 3902 = custom flow sensor 2, 3903 = custom flow sensor 3)
		iSensorTypePort7			: INT;						// ID of the sensor type, that is connected to the port 7 (0 = no sensor, 2001 = SDAP-MHS-M50, 2002 = SDAP-MHS-M100, 2003 = SDAP-MHS-M160, 2901 = custom position sensor 1, 2902 = custom position sensor 2, 2903 = custom position sensor 3, 3001 = SFAB-50U-…-2SA-…, 3002 = SFAB-200U-…-2SA-…, 3003 = SFAB-600U-…-2SA-…, 3004 = SFAB-1000U-…-2SA-…, 3101 = SFAH-50U-…-PNVBA-…, 3102 = SFAH-100U-…-PNVBA-…, 3103 = SFAH-200U-…-PNVBA-…, 3901 = custom flow sensor 1, 3902 = custom flow sensor 2, 3903 = custom flow sensor 3)
		
	// function block response
		iResponse 					: eTransferResponse; 		// returns the status of the upload process
		xBusy						: BOOL;						// TRUE as long as the upload process is running
		xDone 						: BOOL; 					// indicates whether the upload was successfull
		xError 						: BOOL; 					// indicates whether an error occurred during the transfer
		xAborted					: BOOL;						// TRUE if the function block was canceled by xAbort	
END_VAR

VAR
	iState							: INT := 10;
	xStateChange					: BOOL;
	iCommandNumber					: INT;
	xFirstCycle						: BOOL := TRUE;				// indicator for the first cycle of the function block
	iInputModuleNrFC				: INT;						// value on input iInputModuleNr during first cycle
	
	aTransferPackages				: ARRAY [0..100] OF stTransferPackage;
	fbreadbitsfromword				: FB_Read_Bits_From_Word;
	fbuploadMultipleParameters 		: FB_Upload_Multiple_Parameters;
	fbWriteValueToWord 				: FB_Write_Value_To_Word;

	iCounterResetArray				: INT;

	iCurrentValveMode				: INT;						//
END_VAR

(*****************************************************************************************************

Festo SE & Co. KG, Esslingen
Copyright (c) 2021. All rights reserved.

Product:            Motion Terminal VTEM
Description:        Function block to upload the digital module parameters from the Motion Terminal

Object version:     2.00
Last change:        2021-07
======================================================================================================
                                       H I S T O R Y
======================================================================================================
Version:            2.00
Date:               2021-07
Change/Activity:    - created (#3872357)
Release:            3.5.7.237 (CODESYS 3.5.7.2, Lib version 3.7)
Author:             JEBU
======================================================================================================

*****************************************************************************************************)

// pre-check of the value for the parameter set
	IF xExecute = TRUE AND (iInputModuleNr < 1 OR iInputModuleNr > 2) THEN		// invalid input for the module number
		xDone := FALSE; 
		xError := TRUE; 
		iResponse := eTransferResponse.invalid_module_number;
		xStateChange := TRUE;
		iState := 70;	// ERROR
	END_IF
//-----------------------------------------------------------------------------------------------------------

// check if iInputModuleNr was changed
	IF xExecute = TRUE AND xFirstCycle = TRUE THEN
		xFirstCycle := FALSE;
		iInputModuleNrFC := iInputModuleNr;
	END_IF
	
	IF xExecute = TRUE AND iInputModuleNr <> iInputModuleNrFC THEN
		xStateChange := TRUE;
		iState := 70;
		iResponse := eTransferResponse.FB_needs_rising_edge_xExecute;
	END_IF
//-----------------------------------------------------------------------------------------------------------

// WRITE PARAMETER INDICES INTO ARRAY
	// ID of sensor at port 0
		aTransferPackages[0].iChannel := 16;
		aTransferPackages[0].iAddressedTarget := iInputModuleNr;
		aTransferPackages[0].iIndex := 1;
	
	// ID of sensor at port 1
		aTransferPackages[1].iChannel := 16;
		aTransferPackages[1].iAddressedTarget := iInputModuleNr;
		aTransferPackages[1].iIndex := 31;
		
	// ID of sensor at port 2
		aTransferPackages[2].iChannel := 16;
		aTransferPackages[2].iAddressedTarget := iInputModuleNr;
		aTransferPackages[2].iIndex := 61;
    
	// ID of sensor at port 3
		aTransferPackages[3].iChannel := 16;
		aTransferPackages[3].iAddressedTarget := iInputModuleNr;
		aTransferPackages[3].iIndex := 91;
	
	// ID of sensor at port 4
		aTransferPackages[4].iChannel := 16;
		aTransferPackages[4].iAddressedTarget := iInputModuleNr;
		aTransferPackages[4].iIndex := 121;
		
	// ID of sensor at port 5
		aTransferPackages[5].iChannel := 16;
		aTransferPackages[5].iAddressedTarget := iInputModuleNr;
		aTransferPackages[5].iIndex := 151;
			
	// ID of sensor at port 6
		aTransferPackages[6].iChannel := 16;
		aTransferPackages[6].iAddressedTarget := iInputModuleNr;
		aTransferPackages[6].iIndex := 181;
		
	// ID of sensor at port 7
		aTransferPackages[7].iChannel := 16;
		aTransferPackages[7].iAddressedTarget := iInputModuleNr;
		aTransferPackages[7].iIndex := 211;
		
	// define end of parameter list to be uploaded by setting all variables to 0 (end criterion for FB_Upload_Multiple_Parameters)
		aTransferPackages[8].iChannel := 0;
		aTransferPackages[8].iAddressedTarget := 0;
		aTransferPackages[8].iIndex := 0;
//-----------------------------------------------------------------------------------------------------------

// Read the current status of the the motion terminal
	fbreadbitsfromword(wData:= awBusDataFromVTEM[0], iStartBit:=0, iEndBit:= 5, iValue=> iCurrentValveMode, xError=> );				// read current valve mode
//-----------------------------------------------------------------------------------------------------------

// Transition: Aborting condition when xAbort is TRUE in all States except "IDLE" , "ABORTING" and "RESETTING"
	IF xAbort = TRUE AND NOT(iState = 10 AND xExecute = FALSE) AND iState <> 80 AND iState <> 100 THEN
		xStateChange := TRUE;	// Leaving current state
		iState := 80;	// Choosing next state, here: ABORTING
	END_IF
//-----------------------------------------------------------------------------------------------------------

// local state machine
	CASE iState OF
		10:	// IDLE
			// code that is executed only in the first cycle of this state
				IF xStateChange = TRUE THEN
					xStateChange := FALSE;
					iResponse := eTransferResponse.ready_for_new_transfer;
					xDone := FALSE;
					xError := FALSE;
					xBusy := FALSE;
					xAborted := FALSE;
				END_IF
			//-----------------------------------------------------------------------------------------------------------
			
			// code that is repeated every cycle in this state
				iCommandNumber := 0;
			//-----------------------------------------------------------------------------------------------------------
			
			// Transition
			IF xExecute = TRUE THEN
				xStateChange := TRUE;
				iState := 20;
			END_IF
			//-----------------------------------------------------------------------------------------------------------
		
		20:	// RESETTING VALVE MODE TO 61
			// code that is executed only in the first cycle of this state
				IF xStateChange = TRUE THEN
					xStateChange := FALSE;
					iResponse := eTransferResponse.preparing_transfer;
					xDone := FALSE;
					xError := FALSE;
					xBusy := TRUE;
					xAborted := FALSE;
				END_IF
			//-----------------------------------------------------------------------------------------------------------
			
			// code that is repeated every cycle in this state	
				IF iCurrentValveMode = 63 THEN
					iCommandNumber := 5;	// exit transfer mode
				ELSIF iCurrentValveMode <> 61 AND iCurrentValveMode <> 63 THEN
					iCommandNumber := 6;	// stop running motion apps
				END_IF 
			//-----------------------------------------------------------------------------------------------------------
			
			// Transition
				IF iCurrentValveMode = 61 THEN
					xStateChange := TRUE;	// Leave this state
					iState := 30;
					iCommandNumber := 30;			
				END_IF
			//-----------------------------------------------------------------------------------------------------------
		
		30:	// READING PARAMETER VALUES
			// code that is executed only in the first cycle of this state
				IF xStateChange = TRUE THEN
					xStateChange := FALSE;
					iResponse := eTransferResponse.transferring;
					xDone := FALSE;
					xError := FALSE;
					xBusy := TRUE;
					xAborted := FALSE;
				END_IF
			//-----------------------------------------------------------------------------------------------------------
			
			// code that is repeated every cycle in this state
				iCommandNumber := 30;		// read parameter values
			//-----------------------------------------------------------------------------------------------------------
			
			// Transition
				IF fbuploadMultipleParameters.xExecute = TRUE AND fbuploadMultipleParameters.xUploadDone = TRUE AND fbuploadMultipleParameters.xUploadError = FALSE THEN	// Upload Done
					xStateChange := TRUE;
					iState := 40;	// Write parameter values to outputs
				ELSIF fbuploadMultipleParameters.xExecute = TRUE AND fbuploadMultipleParameters.xUploadDone = FALSE AND fbuploadMultipleParameters.xUploadError = TRUE THEN	// Error during update
					xStateChange := TRUE;
					iState := 70;	// ERROR
					iResponse := fbuploadMultipleParameters.iResponse;
				END_IF
			//-----------------------------------------------------------------------------------------------------------
		
		40:	// WRITE PARAMETER VALUES TO OUTPUTS
			// code that is executed only in the first cycle of this state
				IF xStateChange = TRUE THEN
					xStateChange := FALSE;
					iResponse := eTransferResponse.transferring;
					xDone := FALSE;
					xError := FALSE;
					xBusy := TRUE;
					xAborted := FALSE;
				END_IF
			//-----------------------------------------------------------------------------------------------------------
			
			// code that is repeated every cycle in this state
				iSensorTypePort0 := aTransferPackages[0].iTransferValue;
				iSensorTypePort1 := aTransferPackages[1].iTransferValue;
				iSensorTypePort2 := aTransferPackages[2].iTransferValue;
				iSensorTypePort3 := aTransferPackages[3].iTransferValue;
				iSensorTypePort4 := aTransferPackages[4].iTransferValue;
				iSensorTypePort5 := aTransferPackages[5].iTransferValue;
				iSensorTypePort6 := aTransferPackages[6].iTransferValue;
				iSensorTypePort7 := aTransferPackages[7].iTransferValue;
			//-----------------------------------------------------------------------------------------------------------
			
			// Transition
				xStateChange := TRUE;
				iState := 50;
				iCommandNumber := 40;
			//-----------------------------------------------------------------------------------------------------------
		
		50:	// DONE
			// code that is executed only in the first cycle of this state
				IF xStateChange = TRUE THEN
					xStateChange := FALSE;
					iResponse := eTransferResponse.transfer_successful;
					xDone := TRUE;
					xError := FALSE;
					xBusy := FALSE;
					xAborted := FALSE;
				END_IF
			//-----------------------------------------------------------------------------------------------------------
			
			// code that is repeated every cycle in this state	
				IF fbuploadMultipleParameters.xExecute = FALSE  AND fbuploadMultipleParameters.xUploadDone = FALSE AND fbuploadMultipleParameters.xUploadError = FALSE AND iCurrentValveMode = 63 THEN		//FB_UploadMultipleParameters was reset
					iCommandNumber := 5;	// exit transfer mode
				END_IF
			//-----------------------------------------------------------------------------------------------------------
			
			// Transition
				IF fbuploadMultipleParameters.xExecute = FALSE  AND fbuploadMultipleParameters.xUploadDone = FALSE AND fbuploadMultipleParameters.xUploadError = FALSE AND xExecute = FALSE THEN
					xStateChange := TRUE;
					iState := 100;
				END_IF
			//-----------------------------------------------------------------------------------------------------------
			
		70:	// ERROR
			// code that is executed only in the first cycle of this state
				IF xStateChange = TRUE THEN
					xStateChange := FALSE;
					//iResponse := ;	// set within the transition of the last state
					xDone := FALSE;
					xError := TRUE;
					xBusy := FALSE;
					xAborted := FALSE;
				END_IF
			//-----------------------------------------------------------------------------------------------------------
			
			// code that is repeated every cycle in this state	
				IF iResponse = eTransferResponse.invalid_Index THEN
					iResponse := eTransferResponse.invalid_module_number;
				END_IF
			//-----------------------------------------------------------------------------------------------------------
			
			// Transition
				IF xExecute = FALSE AND xAbort = FALSE THEN
					xStateChange := TRUE;
					iState := 100;
				END_IF
			//-----------------------------------------------------------------------------------------------------------
			
		80:	// ABORTING
			// code that is executed only in the first cycle of this state
				IF xStateChange = TRUE THEN
					xStateChange := FALSE;
					iResponse := eTransferResponse.aborting;
					xBusy := FALSE;
					xDone := FALSE;
					xError := FALSE;
					xAborted := TRUE;
				END_IF
			//-----------------------------------------------------------------------------------------------------------
			
			// code that is repeated every cycle in this state
				IF iCurrentValveMode = 63 THEN
					iCommandNumber := 5;	// exit transfer mode
				ELSIF iCurrentValveMode <> 61 AND iCurrentValveMode <> 63 THEN
					iCommandNumber := 6;	// stop running motion apps
				ELSE
					iCommandNumber := 0; 
				END_IF
			//-----------------------------------------------------------------------------------------------------------
			
			// Transition
				IF xAbort = FALSE AND xExecute = FALSE AND iCurrentValveMode = 61 THEN
					xStateChange := TRUE;
					iState := 100;
				END_IF
			//-----------------------------------------------------------------------------------------------------------

		100:	// RESETTING FUNCTION BLOCK AND VALVE
			// code that is executed only in the first cycle of this state
				IF xStateChange = TRUE THEN
					xStateChange := FALSE;
					iResponse := eTransferResponse.resetting;
					xDone := FALSE;
					xError := FALSE;
					xBusy := FALSE;
					xAborted := FALSE;
				END_IF
			//-----------------------------------------------------------------------------------------------------------
			
			// code that is repeated every cycle in this state	
				IF iCurrentValveMode = 63 THEN
					iCommandNumber := 5;	// exit transfer mode
				ELSIF iCurrentValveMode <> 61 AND iCurrentValveMode <> 63 THEN
					iCommandNumber := 6;	// stop running motion apps
				END_IF
				
				// reset funktion block fbreadmultipleparameters
				// not done via command number because this is used to reset valve
					fbuploadMultipleParameters(
						awBusDataFromVTEM:= awBusDataFromVTEM, 
						awBusDataToVTEM:= awBusDataToVTEM, 
						xExecute:= FALSE, 
						iResponse=> , 
						iCurrentValue=> , 
						xUploadDone=> , 
						xUploadError=> , 
						aTransferPackages:= aTransferPackages);
				
				// reset parameter outputs
					iInputModuleNr			:= 0;

					iSensorTypePort0		:= 0;
					iSensorTypePort1		:= 0;
					iSensorTypePort2		:= 0;
					iSensorTypePort3		:= 0;
					iSensorTypePort4		:= 0;
					iSensorTypePort5		:= 0;
					iSensorTypePort6		:= 0;
					iSensorTypePort7		:= 0;
				
				// reset parameter array
					FOR iCounterResetArray := 0 TO 100 BY 1 DO
						aTransferPackages[iCounterResetArray].iChannel := 0;
						aTransferPackages[iCounterResetArray].iAddressedTarget := 0;
						aTransferPackages[iCounterResetArray].iIndex := 0;
						aTransferPackages[iCounterResetArray].iTransferValue := 0;
					END_FOR
					
					iCounterResetArray := 0;
					xFirstCycle := TRUE;
			//-----------------------------------------------------------------------------------------------------------
			
			// Transition
				IF iCurrentValveMode = 61 THEN
					iCommandNumber := 6; // Last command to send before the FB is in IDLE
					xStateChange := TRUE;
					iState := 10;
				END_IF
			//-----------------------------------------------------------------------------------------------------------
			
	END_CASE
//-----------------------------------------------------------------------------------------------------------

// Command section
	CASE iCommandNumber OF
		0:	// IDLE
			;
		
		5:	// EXIT TRANSFER MODE
			fbwritevaluetoword(iValue:=63, iStartBit:=0, iEndBit:=5, wDataWord:=awBusDataToVTEM[0], xError=> );							// Valve Mode = 63
			fbwritevaluetoword(iValue:=0, iStartBit:=6, iEndBit:=7, wDataWord:=awBusDataToVTEM[0], xError=> );							// 0 (unused)
			fbwritevaluetoword(iValue:=0, iStartBit:=8, iEndBit:=12, wDataWord:=awBusDataToVTEM[0], xError=> );							// Channel = 0 (ignored)
			fbwritevaluetoword(iValue:=3, iStartBit:=13, iEndBit:=15, wDataWord:=awBusDataToVTEM[0], xError=> );						// Transfer Control = 3 (Exit transfer mode)
			fbwritevaluetoword(iValue:=0, iStartBit:=0, iEndBit:=7, wDataWord:=awBusDataToVTEM[1], xError=> );							// Addressed Target = 0 (ignored)
			fbwritevaluetoword(iValue:=0, iStartBit:=8, iEndBit:=15, wDataWord:=awBusDataToVTEM[1], xError=> );							// Index = 0 (ignored)
			fbwritevaluetoword(iValue:=0, iStartBit:=0, iEndBit:=15, wDataWord:=awBusDataToVTEM[2], xError=> );							// Value = 0 (ignored)
			
		6:	// STOP RUNNING MOTION APP
			fbwritevaluetoword(iValue:=61, iStartBit:=0, iEndBit:=5, wDataWord:=awBusDataToVTEM[0], xError=> );							// Valve Mode = 61 (stop)
			fbwritevaluetoword(iValue:=0, iStartBit:=6, iEndBit:=7, wDataWord:=awBusDataToVTEM[0], xError=> );							// App Control = 0 (unused)
			fbwritevaluetoword(iValue:=0, iStartBit:=8, iEndBit:=15, wDataWord:=awBusDataToVTEM[0], xError=> );							// App Option = 0 (unused)
			fbwritevaluetoword(iValue:=0, iStartBit:=0, iEndBit:=15, wDataWord:=awBusDataToVTEM[1], xError=> );							// Setpoint Value 1 = 0 (unused)
			fbwritevaluetoword(iValue:=0, iStartBit:=0, iEndBit:=15, wDataWord:=awBusDataToVTEM[2], xError=> );							// Setpoint Value 2 = 0 (unused)
		
		30:	// RUN FB_UPLOADMULTIPLEPARAMETERS
			fbuploadMultipleParameters(
				awBusDataFromVTEM:= awBusDataFromVTEM, 
				awBusDataToVTEM:= awBusDataToVTEM, 
				xExecute:= TRUE, 
				iResponse=> , 
				iCurrentValue=> , 
				xUploadDone=> , 
				xUploadError=> , 
				aTransferPackages:= aTransferPackages);

		40:	// RESET FB_UPLOADMULTIPLEPARAMETERS
			fbuploadMultipleParameters(
				awBusDataFromVTEM:= awBusDataFromVTEM, 
				awBusDataToVTEM:= awBusDataToVTEM, 
				xExecute:= FALSE, 
				iResponse=> , 
				iCurrentValue=> , 
				xUploadDone=> , 
				xUploadError=> , 
				aTransferPackages:= aTransferPackages);
	END_CASE
//-----------------------------------------------------------------------------------------------------------

END_FUNCTION_BLOCK
